# EPICS StreamDevice protocol: sorensenPS/proto/test.proto
#terminator = CR LF;

read {
    out "%s";
    in "%s";
}
